// TIA Portal project "4M - 1" (V16)

(* hardware
DEVICE "S7-1200 station_1"  S7-1200 Station
   slot 0: "Rack_0"  S7-1200 Rack  Rack  V1.0
   slot 1: "PLC_1"  CPU 1212C AC/DC/Rly  6ES7 212-1BE40-0XB0  V4.0
*)

// ===== PLC "PLC_1"  CPU 1212C AC/DC/Rly =====

VAR_GLOBAL   // PLC tag table "Default tag table"
   "K1" AT %Q0.0 : Bool;
   "stop1" AT %I0.4 : Bool;
   "k2" AT %Q0.1 : Bool;
   "X" AT %M0.0 : Bool;
   "K3" AT %Q0.2 : Bool;
   "start1" AT %I0.2 : Bool;
   "c1" AT %M0.1 : Bool;
   "c3" AT %M0.3 : Bool;
   "c4" AT %M0.4 : Bool;
   "Tag_5" AT %M1.1 : Bool;
   "t4 tag" AT %M1.0 : Bool;
   "t1 tag" AT %M0.5 : Bool;
   "k4" AT %Q0.3 : Bool;
   "c2" AT %M0.2 : Bool;
   "t2 tag" AT %M0.6 : Bool;
   "t3 tag" AT %M0.7 : Bool;
   "STOP" AT %I0.3 : Bool;
END_VAR

// folder: System blocks/Program resources

DATA_BLOCK "T4"   // DB1
{ S7_Optimized_Access := 'TRUE' }
AUTHOR : Simatic
FAMILY : IEC
NAME : IEC_TMR
VERSION : 1.0
// stored: InstanceOfName IEC_TIMER
"IEC_TIMER"
BEGIN
END_DATA_BLOCK

DATA_BLOCK "T1"   // DB2
{ S7_Optimized_Access := 'TRUE' }
AUTHOR : Simatic
FAMILY : IEC
NAME : IEC_TMR
VERSION : 1.0
// stored: InstanceOfName IEC_TIMER
"IEC_TIMER"
BEGIN
END_DATA_BLOCK

DATA_BLOCK "T2"   // DB3
{ S7_Optimized_Access := 'TRUE' }
AUTHOR : Simatic
FAMILY : IEC
NAME : IEC_TMR
VERSION : 1.0
// stored: InstanceOfName IEC_TIMER
"IEC_TIMER"
BEGIN
END_DATA_BLOCK

DATA_BLOCK "T3"   // DB4
{ S7_Optimized_Access := 'TRUE' }
AUTHOR : Simatic
FAMILY : IEC
NAME : IEC_TMR
VERSION : 1.0
// stored: InstanceOfName IEC_TIMER
"IEC_TIMER"
BEGIN
END_DATA_BLOCK

// folder: (top level)

ORGANIZATION_BLOCK "Main"   // OB1, LAD, ProgramCycle
TITLE = "Main Program Sweep (Cycle)"
{ S7_Optimized_Access := 'TRUE' }
VERSION : 0.1
   VAR_INPUT
      Initial_Call : Bool;   // Initial call of this OB
      Remanence : Bool;   // =True, if remanent data are available
   END_VAR
BEGIN

REGION Network 1: start
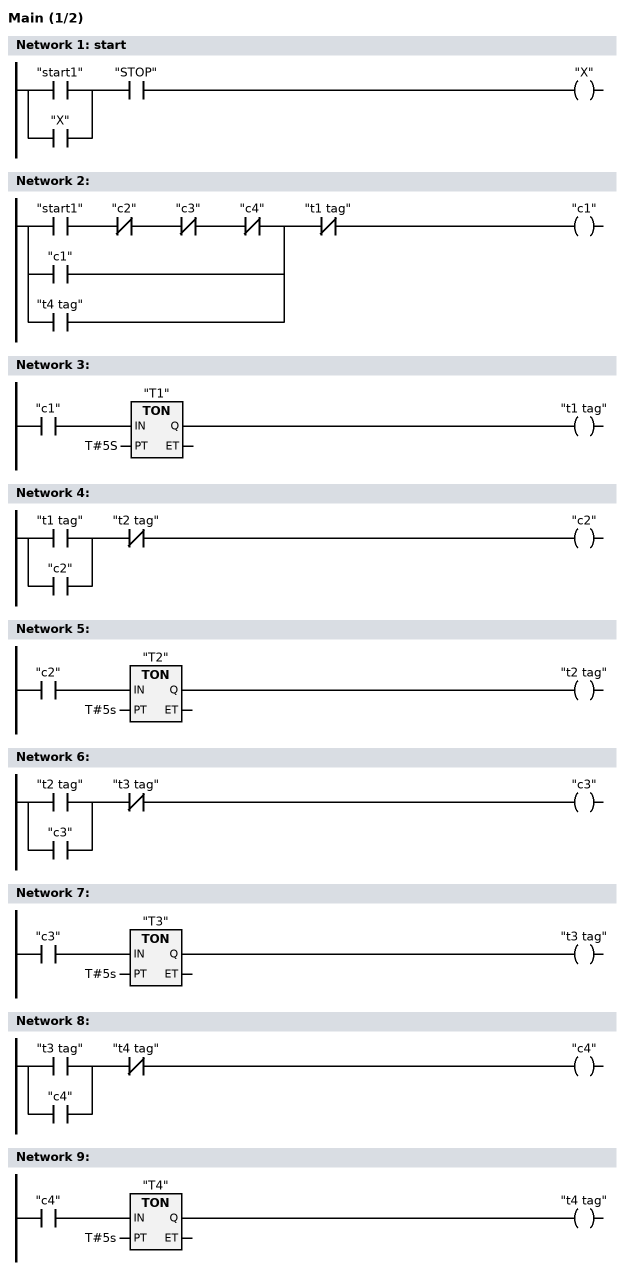
   RUNG wire#powerrail
      Contact( "start1" )
      wire#w1
      Contact( "STOP" )
      Coil( "X" )
   END_RUNG
   RUNG wire#powerrail
      Contact( "X" )
   END_RUNG wire#w1
   // the same network as SCL:
   "X" := ("start1" OR "X") AND "STOP";
END_REGION

REGION Network 2
   RUNG wire#powerrail
      Contact( "start1" )
      I_Contact( "c2" )
      I_Contact( "c3" )
      I_Contact( "c4" )
      wire#w1
      I_Contact( "t1 tag" )
      Coil( "c1" )
   END_RUNG
   RUNG wire#powerrail
      Contact( "c1" )
   END_RUNG wire#w1
   RUNG wire#powerrail
      Contact( "t4 tag" )
   END_RUNG wire#w1
   // the same network as SCL:
   "c1" := (("start1" AND NOT "c2" AND NOT "c3" AND NOT "c4") OR "c1" OR "t4 tag") AND NOT "t1 tag";
END_REGION

REGION Network 3
   "T1".TON(IN := "c1", PT := T#5S);
   "t1 tag" := "T1".Q;
END_REGION

REGION Network 4
   RUNG wire#powerrail
      Contact( "t1 tag" )
      wire#w1
      I_Contact( "t2 tag" )
      Coil( "c2" )
   END_RUNG
   RUNG wire#powerrail
      Contact( "c2" )
   END_RUNG wire#w1
   // the same network as SCL:
   "c2" := ("t1 tag" OR "c2") AND NOT "t2 tag";
END_REGION

REGION Network 5
   "T2".TON(IN := "c2", PT := T#5s);
   "t2 tag" := "T2".Q;
END_REGION

REGION Network 6
   RUNG wire#powerrail
      Contact( "t2 tag" )
      wire#w1
      I_Contact( "t3 tag" )
      Coil( "c3" )
   END_RUNG
   RUNG wire#powerrail
      Contact( "c3" )
   END_RUNG wire#w1
   // the same network as SCL:
   "c3" := ("t2 tag" OR "c3") AND NOT "t3 tag";
END_REGION

REGION Network 7
   "T3".TON(IN := "c3", PT := T#5s);
   "t3 tag" := "T3".Q;
END_REGION

REGION Network 8
   RUNG wire#powerrail
      Contact( "t3 tag" )
      wire#w1
      I_Contact( "t4 tag" )
      Coil( "c4" )
   END_RUNG
   RUNG wire#powerrail
      Contact( "c4" )
   END_RUNG wire#w1
   // the same network as SCL:
   "c4" := ("t3 tag" OR "c4") AND NOT "t4 tag";
END_REGION

REGION Network 9
   "T4".TON(IN := "c4", PT := T#5s);
   "t4 tag" := "T4".Q;
END_REGION

REGION Network 10
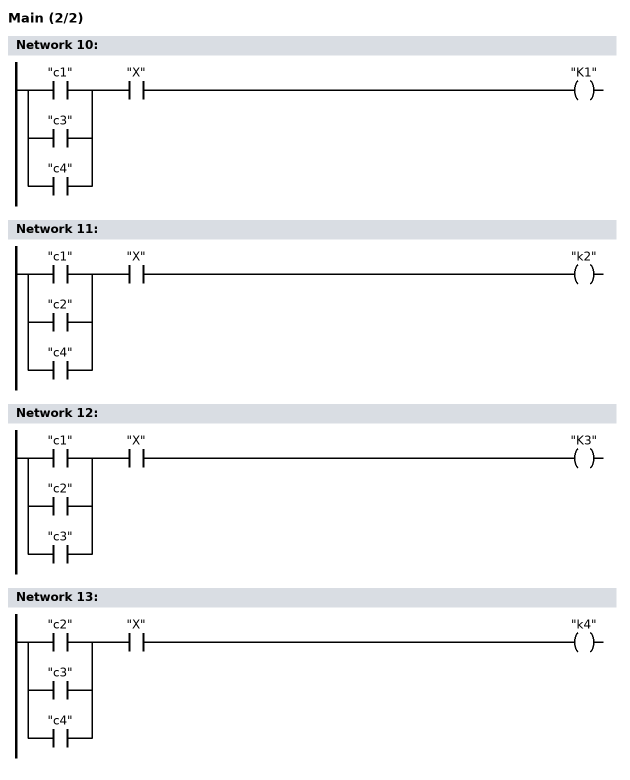
   RUNG wire#powerrail
      Contact( "c1" )
      wire#w1
      Contact( "X" )
      Coil( "K1" )
   END_RUNG
   RUNG wire#powerrail
      Contact( "c3" )
   END_RUNG wire#w1
   RUNG wire#powerrail
      Contact( "c4" )
   END_RUNG wire#w1
   // the same network as SCL:
   "K1" := ("c1" OR "c3" OR "c4") AND "X";
END_REGION

REGION Network 11
   RUNG wire#powerrail
      Contact( "c1" )
      wire#w1
      Contact( "X" )
      Coil( "k2" )
   END_RUNG
   RUNG wire#powerrail
      Contact( "c2" )
   END_RUNG wire#w1
   RUNG wire#powerrail
      Contact( "c4" )
   END_RUNG wire#w1
   // the same network as SCL:
   "k2" := ("c1" OR "c2" OR "c4") AND "X";
END_REGION

REGION Network 12
   RUNG wire#powerrail
      Contact( "c1" )
      wire#w1
      Contact( "X" )
      Coil( "K3" )
   END_RUNG
   RUNG wire#powerrail
      Contact( "c2" )
   END_RUNG wire#w1
   RUNG wire#powerrail
      Contact( "c3" )
   END_RUNG wire#w1
   // the same network as SCL:
   "K3" := ("c1" OR "c2" OR "c3") AND "X";
END_REGION

REGION Network 13
   RUNG wire#powerrail
      Contact( "c2" )
      wire#w1
      Contact( "X" )
      Coil( "k4" )
   END_RUNG
   RUNG wire#powerrail
      Contact( "c3" )
   END_RUNG wire#w1
   RUNG wire#powerrail
      Contact( "c4" )
   END_RUNG wire#w1
   // the same network as SCL:
   "k4" := ("c2" OR "c3" OR "c4") AND "X";
END_REGION
END_ORGANIZATION_BLOCK